                    // ---------- LT2100E register unpack (HMI writes %MW600..609) ----------
// reg[0] button bits: 0=start 1=stop 2=reset 3=ack 4=clean
//                     5=jog+ 6=jog- 7=recipeWrite 8=trimWrite
// Numerics are copied only while their write/jog bit is held, so direct
// variable writes (watch list / sim testing) keep working unchanged.
IF GVL_Cmd.hmiRegsCmd[1] <> 0 THEN
    GVL_Cmd.hmiMaintPin := TO_UINT(GVL_Cmd.hmiRegsCmd[1]);
END_IF
IF (GVL_Cmd.hmiRegsCmd[0] AND 16#0060) <> 0 THEN            // a jog bit is held
    GVL_Cmd.hmiJogAxis := TO_INT(GVL_Cmd.hmiRegsCmd[2]);
END_IF
IF (GVL_Cmd.hmiRegsCmd[0] AND 16#0080) <> 0 THEN            // recipe write
    GVL_Cmd.hmiRecItem  := TO_UINT(GVL_Cmd.hmiRegsCmd[3]);
    GVL_Cmd.hmiRecField := TO_UINT(GVL_Cmd.hmiRegsCmd[4]);
    GVL_Cmd.hmiRecValue := TO_LREAL(GVL_Cmd.hmiRegsCmd[5]) / 10.0;   // x10 scaling
END_IF
IF (GVL_Cmd.hmiRegsCmd[0] AND 16#0100) <> 0 THEN            // trim write
    GVL_Cmd.hmiTrimPress := TO_UINT(GVL_Cmd.hmiRegsCmd[6]);
    GVL_Cmd.hmiTrimDelta := TO_LREAL(TO_INT(GVL_Cmd.hmiRegsCmd[7])) / 100.0;  // x100 signed
END_IF
bJogP := GVL_Cmd.hmiJogPlus  OR ((GVL_Cmd.hmiRegsCmd[0] AND 16#0020) <> 0);
bJogM := GVL_Cmd.hmiJogMinus OR ((GVL_Cmd.hmiRegsCmd[0] AND 16#0040) <> 0);

rtStart(CLK := GVL_Cmd.hmiStart OR ((GVL_Cmd.hmiRegsCmd[0] AND 16#0001) <> 0));
rtStop (CLK := GVL_Cmd.hmiStop  OR ((GVL_Cmd.hmiRegsCmd[0] AND 16#0002) <> 0));
rtReset(CLK := GVL_Cmd.hmiReset OR ((GVL_Cmd.hmiRegsCmd[0] AND 16#0004) <> 0));
rtAck  (CLK := GVL_Cmd.hmiAck   OR ((GVL_Cmd.hmiRegsCmd[0] AND 16#0008) <> 0));
rtClean(CLK := GVL_Cmd.hmiClean OR ((GVL_Cmd.hmiRegsCmd[0] AND 16#0010) <> 0));

GVL_Cmd.reqStart  := rtStart.Q;
GVL_Cmd.reqStop   := rtStop.Q  OR GVL_Cmd.reqStop;    // JobExec may also set; consumed by Supervisor edge
GVL_Cmd.reqReset  := rtReset.Q;
GVL_Cmd.reqAckAll := rtAck.Q;
GVL_Cmd.reqClean  := rtClean.Q OR GVL_Cmd.reqClean;
// self-clearing one-shot semantics: Supervisor uses R_TRIG on these,
// so clear them after one comms cycle
IF NOT rtStop.Q  THEN GVL_Cmd.reqStop  := FALSE; END_IF
IF NOT rtClean.Q THEN GVL_Cmd.reqClean := FALSE; END_IF

// ---------- jog (maintenance only) ----------
jogPermit := (GVL_Cmd.hmiMaintPin = MAINT_PIN)
         AND ((GVL_Sts.mode = E_MachMode.READY) OR (GVL_Sts.mode = E_MachMode.FAULT))
         AND GVL_Sts.safetyOk;
tonJog(IN := jogPermit AND (bJogP OR bJogM), PT := T#100MS);
IF tonJog.Q THEN
    tonJog(IN := FALSE);
    jogStep := LIMIT(1.0, GVL_Par.jogVel, GVL_Cfg.JOG_VEL_MAX) * 0.1;  // mm per 100 ms
    IF bJogM THEN jogStep := -jogStep; END_IF
    CASE GVL_Cmd.hmiJogAxis OF
        1: IF NOT GVL_Mech.axGX.Busy THEN
               GVL_Mech.axGX.TargetPos := GVL_Mech.axGX.Sts.actPos + jogStep;
               GVL_Mech.axGX.Vel := GVL_Par.jogVel;
               GVL_Mech.axGX.MoveExec := TRUE;
           END_IF
        2: IF NOT GVL_Mech.axGT.Busy THEN
               GVL_Mech.axGT.TargetPos := GVL_Mech.axGT.Sts.actPos + jogStep;
               GVL_Mech.axGT.Vel := GVL_Par.jogVel;
               GVL_Mech.axGT.MoveExec := TRUE;
           END_IF
        3: IF NOT GVL_Mech.axGZ.Busy THEN
               GVL_Mech.axGZ.TargetPos := GVL_Mech.axGZ.Sts.actPos + jogStep;
               GVL_Mech.axGZ.Vel := GVL_Par.jogVel;
               GVL_Mech.axGZ.MoveExec := TRUE;
           END_IF
        // axes 4..8: same pattern for scraper X/Y/Z, fork Z/tele — add as needed
    END_CASE
ELSIF NOT (bJogP OR bJogM) THEN
    GVL_Mech.axGX.MoveExec := FALSE;
    GVL_Mech.axGT.MoveExec := FALSE;
    GVL_Mech.axGZ.MoveExec := FALSE;
END_IF

// ---------- recipe editor (bounds-checked; rejected while RUN) ----------
rtRecW(CLK := GVL_Cmd.hmiRecWrite OR ((GVL_Cmd.hmiRegsCmd[0] AND 16#0080) <> 0));
IF rtRecW.Q THEN
    GVL_Cmd.hmiRecAck := FALSE; GVL_Cmd.hmiRecErr := FALSE;
    recIt := TO_INT(GVL_Cmd.hmiRecItem);
    recV  := GVL_Cmd.hmiRecValue;
    recOk := (recIt >= 1) AND (recIt <= 4) AND (GVL_Sts.mode <> E_MachMode.RUN);
    IF recOk THEN
        CASE GVL_Cmd.hmiRecField OF
            1: IF (recV >= GVL_Cfg.REC_COOK_MIN)  AND (recV <= GVL_Cfg.REC_COOK_MAX)
               THEN GVL_Par.aRecipe[recIt].cookTimeS := recV;  ELSE recOk := FALSE; END_IF
            2: IF (recV >= GVL_Cfg.REC_SMDUR_MIN) AND (recV <= GVL_Cfg.REC_SMDUR_MAX)
               THEN GVL_Par.aRecipe[recIt].smashDurS := recV;  ELSE recOk := FALSE; END_IF
            3: IF (recV >= GVL_Cfg.REC_SMPOS_MIN) AND (recV <= GVL_Cfg.REC_SMPOS_MAX)
               THEN GVL_Par.aRecipe[recIt].smashPosMm := recV; ELSE recOk := FALSE; END_IF
            4: IF (recV >= GVL_Cfg.REC_HLPOS_MIN) AND (recV <= GVL_Cfg.REC_HLPOS_MAX)
               THEN GVL_Par.aRecipe[recIt].holdPosMm := recV;  ELSE recOk := FALSE; END_IF
            5: IF (recV >= GVL_Cfg.REC_PLSET_MIN) AND (recV <= GVL_Cfg.REC_PLSET_MAX)
               THEN GVL_Par.aRecipe[recIt].platenSetC := recV; ELSE recOk := FALSE; END_IF
        ELSE
            recOk := FALSE;
        END_CASE
        // physical sanity: hold gap must not be tighter than smash gap
        IF recOk AND (GVL_Par.aRecipe[recIt].holdPosMm < GVL_Par.aRecipe[recIt].smashPosMm) THEN
            GVL_Par.aRecipe[recIt].holdPosMm := GVL_Par.aRecipe[recIt].smashPosMm;
        END_IF
    END_IF
    GVL_Cmd.hmiRecAck := recOk;
    GVL_Cmd.hmiRecErr := NOT recOk;
END_IF

// ---------- press calibration trim (maintenance PIN; not while RUN) ----------
rtTrimW(CLK := GVL_Cmd.hmiTrimWrite OR ((GVL_Cmd.hmiRegsCmd[0] AND 16#0100) <> 0));
IF rtTrimW.Q THEN
    GVL_Cmd.hmiTrimAck := FALSE; GVL_Cmd.hmiTrimErr := FALSE;
    trimP := TO_INT(GVL_Cmd.hmiTrimPress);
    IF (trimP >= 0) AND (trimP <= 3)
       AND (GVL_Cmd.hmiMaintPin = MAINT_PIN)
       AND (GVL_Sts.mode <> E_MachMode.RUN)
       AND (ABS(GVL_Cmd.hmiTrimDelta) <= GVL_Cfg.PRESS_TRIM_MAX_MM) THEN
        GVL_Par.pressTrimMm[trimP] := LIMIT(-GVL_Cfg.PRESS_TRIM_MAX_MM,
            GVL_Par.pressTrimMm[trimP] + GVL_Cmd.hmiTrimDelta,
            GVL_Cfg.PRESS_TRIM_MAX_MM);
        GVL_Cmd.hmiTrimAck := TRUE;
    ELSE
        GVL_Cmd.hmiTrimErr := TRUE;
    END_IF
END_IF

// ---------- LT2100E status pack (HMI reads %MW620..669) ----------
GVL_Cmd.hmiRegsSts[0] := TO_WORD(TO_UINT(GVL_Sts.mode));
wFlags := 0;
IF GVL_Cmd.hmiRecAck    THEN wFlags := wFlags OR 16#0001; END_IF
IF GVL_Cmd.hmiRecErr    THEN wFlags := wFlags OR 16#0002; END_IF
IF GVL_Cmd.hmiTrimAck   THEN wFlags := wFlags OR 16#0004; END_IF
IF GVL_Cmd.hmiTrimErr   THEN wFlags := wFlags OR 16#0008; END_IF
IF GVL_Sts.heatAtSet    THEN wFlags := wFlags OR 16#0010; END_IF
IF GVL_Sts.fridgeAtSet  THEN wFlags := wFlags OR 16#0020; END_IF
IF GVL_Sts.allHomed     THEN wFlags := wFlags OR 16#0040; END_IF
IF GVL_Sts.safetyOk     THEN wFlags := wFlags OR 16#0080; END_IF
IF GVL_Sts.cleanCoolOk  THEN wFlags := wFlags OR 16#0100; END_IF
GVL_Cmd.hmiRegsSts[1] := wFlags;
GVL_Cmd.hmiRegsSts[2] := TO_WORD(TO_UINT(GVL_Alm.nActive));
GVL_Cmd.hmiRegsSts[3] := TO_WORD(GVL_Alm.aActive[0].id AND 16#FFFF);          // code
GVL_Cmd.hmiRegsSts[4] := TO_WORD(SHR(GVL_Alm.aActive[0].id, 16) AND 16#FFFF); // subsystem
GVL_Cmd.hmiRegsSts[5] := TO_WORD(TO_UINT(GVL_Sts.uptimeS MOD 65536));
// griddle states 626..629
FOR z2 := 0 TO 3 DO
    GVL_Cmd.hmiRegsSts[6 + z2] := TO_WORD(GVL_Sts.aGriddle[z2].state);
END_FOR
// recipe readback 630..649: per item 1..4 -> cook, smashDur, smashPos, holdPos, platenSet (all x10)
FOR it2 := 1 TO 4 DO
    base := 10 + (it2 - 1) * 5;
    GVL_Cmd.hmiRegsSts[base]     := TO_WORD(TO_UINT(GVL_Par.aRecipe[it2].cookTimeS  * 10.0));
    GVL_Cmd.hmiRegsSts[base + 1] := TO_WORD(TO_UINT(GVL_Par.aRecipe[it2].smashDurS  * 10.0));
    GVL_Cmd.hmiRegsSts[base + 2] := TO_WORD(TO_UINT(GVL_Par.aRecipe[it2].smashPosMm * 10.0));
    GVL_Cmd.hmiRegsSts[base + 3] := TO_WORD(TO_UINT(GVL_Par.aRecipe[it2].holdPosMm  * 10.0));
    GVL_Cmd.hmiRegsSts[base + 4] := TO_WORD(TO_UINT(GVL_Par.aRecipe[it2].platenSetC * 10.0));
END_FOR
// press trims 650..653 (x100 signed)
FOR z2 := 0 TO 3 DO
    GVL_Cmd.hmiRegsSts[30 + z2] := TO_WORD(TO_INT(GVL_Par.pressTrimMm[z2] * 100.0));
END_FOR
// temperatures 654..661 platens, 662 fridge (x10)
FOR z2 := 0 TO 7 DO
    GVL_Cmd.hmiRegsSts[34 + z2] := TO_WORD(TO_INT(GVL_Sts.aHeat[z2].actC * 10.0));
END_FOR
GVL_Cmd.hmiRegsSts[42] := TO_WORD(TO_INT(GVL_Sts.fridgeActC * 10.0));

                  
END_PROGRAM

(* ============================================================ PRG_Carousels — T_App body-call owner: press drives, presses, pneumatics, VFD indexers, carousels, airlock. Pure wiring (the ST equivalent of a CFC sheet). Runs AFTER Supervisor/ JobExec/Test (which write the Cmd inputs). ============================================================ *)
PROGRAM PRG_Carousels
  VAR
    i : INT;
    init : BOOL;
  END_VAR

                    IF NOT init THEN
    init := TRUE;
    FOR i := 0 TO 3 DO
        GVL_Mech.drvPress[i].SubsysId := GVL_Cfg.SS_PRESS_0 + TO_UINT(i);
        GVL_Mech.fbPress[i].PressId := i;
    END_FOR
    GVL_Mech.fbDoorFridgeFront.SubsysId := GVL_Cfg.SS_AIRLOCK;
    GVL_Mech.fbDoorFridgeSide.SubsysId  := GVL_Cfg.SS_AIRLOCK;
    GVL_Mech.fbDoorChamber.SubsysId     := GVL_Cfg.SS_AIRLOCK;
    GVL_Mech.fbPinGriddle.SubsysId := GVL_Cfg.SS_GRID_CAR;
    GVL_Mech.fbPinFridge.SubsysId  := GVL_Cfg.SS_FRIDGE_CAR;
    GVL_Mech.fbPneuGrip.SubsysId   := GVL_Cfg.SS_GRIPPER;
    GVL_Mech.vfdGriddle.SubsysId := GVL_Cfg.SS_GRID_CAR;
    GVL_Mech.vfdFridge.SubsysId  := GVL_Cfg.SS_FRIDGE_CAR;
END_IF

// ---- presses ----
FOR i := 0 TO 3 DO
    GVL_Mech.fbPress[i].Enable := GVL_Sts.enMotion;
    GVL_Mech.fbPress[i].Abort  := GVL_Sts.abortAll;
    GVL_Mech.fbPress[i].Sim    := GVL_Cfg.SIM_MODE;
    GVL_Mech.fbPress[i].CycleMs:= GVL_Cfg.T_APP_MS;
    // bench override: the selected drive runs REAL while the machine is sim
    GVL_Mech.drvPress[i].Sim    := GVL_Cfg.SIM_MODE AND (i <> GVL_Cfg.PRESS_BENCH_DRIVE);
    GVL_Mech.drvPress[i].Enable := GVL_Sts.enMotion;
    GVL_Mech.drvPress[i].Abort  := GVL_Sts.abortAll;
    GVL_Mech.drvPress[i].CycleMs:= GVL_Cfg.T_APP_MS;
    GVL_Mech.drvPress[i].iInPos := GVL_IO.iPressInPos[i];
    GVL_Mech.drvPress[i].iAlarm := GVL_IO.iPressAlarm[i];
    GVL_Mech.fbPress[i](Drv := GVL_Mech.drvPress[i]);
    GVL_Mech.drvPress[i]();
    IF (NOT GVL_Cfg.SIM_MODE) OR (i = GVL_Cfg.PRESS_BENCH_DRIVE) THEN
        GVL_IO.qPressSel0[i]   := GVL_Mech.drvPress[i].qSel0;
        GVL_IO.qPressSel1[i]   := GVL_Mech.drvPress[i].qSel1;
        GVL_IO.qPressCtrg[i]   := GVL_Mech.drvPress[i].qCtrg;
        GVL_IO.qPressEnable[i] := GVL_Mech.drvPress[i].qEnable;
    END_IF
END_FOR

// ---- CS2RS Modbus PR-write transport: NetworkConfig channel routing ----
// Channels are created in NetworkConfig (RS485 -> Modbus Master), one
// write-multiple channel per PR path (see GVL_IO placeholders + GVL_Cfg
// reference). This glue routes the bench/press-0 drive's path-write request
// to the matching channel. Extend with channel banks for drives 1..3 when
// the full RS485 bus exists.
IF (NOT GVL_Cfg.SIM_MODE) OR (GVL_Cfg.PRESS_BENCH_DRIVE >= 0) THEN
    GVL_IO.qMbPr0Trig := FALSE;
    GVL_IO.qMbPr1Trig := FALSE;
    GVL_IO.qMbPr2Trig := FALSE;
    GVL_Mech.drvPress[0].MbWrDone := FALSE;
    GVL_Mech.drvPress[0].MbWrErr  := FALSE;
    CASE GVL_Mech.drvPress[0].MbPath OF
        0:  GVL_IO.qMbPr0Data[0] := GVL_Mech.drvPress[0].MbValH;
            GVL_IO.qMbPr0Data[1] := GVL_Mech.drvPress[0].MbValL;
            GVL_IO.qMbPr0Trig    := GVL_Mech.drvPress[0].MbWrExec;
            GVL_Mech.drvPress[0].MbWrDone := GVL_IO.iMbPr0Done AND GVL_Mech.drvPress[0].MbWrExec;
        1:  GVL_IO.qMbPr1Data[0] := GVL_Mech.drvPress[0].MbValH;
            GVL_IO.qMbPr1Data[1] := GVL_Mech.drvPress[0].MbValL;
            GVL_IO.qMbPr1Trig    := GVL_Mech.drvPress[0].MbWrExec;
            GVL_Mech.drvPress[0].MbWrDone := GVL_IO.iMbPr1Done AND GVL_Mech.drvPress[0].MbWrExec;
        2:  GVL_IO.qMbPr2Data[0] := GVL_Mech.drvPress[0].MbValH;
            GVL_IO.qMbPr2Data[1] := GVL_Mech.drvPress[0].MbValL;
            GVL_IO.qMbPr2Trig    := GVL_Mech.drvPress[0].MbWrExec;
            GVL_Mech.drvPress[0].MbWrDone := GVL_IO.iMbPr2Done AND GVL_Mech.drvPress[0].MbWrExec;
    END_CASE
    GVL_Mech.drvPress[0].MbWrErr :=
        (GVL_IO.iMbPrErr <> 0) AND GVL_Mech.drvPress[0].MbWrExec;
END_IF

// ---- pneumatics ----
GVL_Mech.fbDoorFridgeSide(Sim := GVL_Cfg.SIM_MODE, CycleMs := GVL_Cfg.T_APP_MS,
    iExtended := GVL_IO.iDoorFrSide_Op, iRetracted := GVL_IO.iDoorFrSide_Cl);
GVL_Mech.fbDoorChamber(Sim := GVL_Cfg.SIM_MODE, CycleMs := GVL_Cfg.T_APP_MS,
    iExtended := GVL_IO.iDoorChamber_Op, iRetracted := GVL_IO.iDoorChamber_Cl);
GVL_Mech.fbDoorFridgeFront(Sim := GVL_Cfg.SIM_MODE, CycleMs := GVL_Cfg.T_APP_MS,
    iExtended := GVL_IO.iDoorFrFront_Op, iRetracted := GVL_IO.iDoorFrFront_Cl);
GVL_Mech.fbPinGriddle(Sim := GVL_Cfg.SIM_MODE, CycleMs := GVL_Cfg.T_APP_MS,
    iExtended := GVL_IO.iPinGriddle_Ext, iRetracted := GVL_IO.iPinGriddle_Ret);
GVL_Mech.fbPinFridge(Sim := GVL_Cfg.SIM_MODE, CycleMs := GVL_Cfg.T_APP_MS,
    iExtended := GVL_IO.iPinFridge_Ext, iRetracted := GVL_IO.iPinFridge_Ret);
GVL_Mech.fbPneuGrip(Sim := GVL_Cfg.SIM_MODE, CycleMs := GVL_Cfg.T_APP_MS,
    iExtended := GVL_IO.iGripAcquired, iRetracted := NOT GVL_IO.iGripAcquired);
IF NOT GVL_Cfg.SIM_MODE THEN
    GVL_IO.qDoorFridgeSide  := GVL_Mech.fbDoorFridgeSide.qValve;
    GVL_IO.qDoorChamber     := GVL_Mech.fbDoorChamber.qValve;
    GVL_IO.qDoorFridgeFront := GVL_Mech.fbDoorFridgeFront.qValve;
    GVL_IO.qPinGriddle      := GVL_Mech.fbPinGriddle.qValve;
    GVL_IO.qPinFridge       := GVL_Mech.fbPinFridge.qValve;
    GVL_IO.qGripper         := GVL_Mech.fbPneuGrip.qValve;
END_IF

// ---- airlock ----
GVL_Mech.fbAirlock(
    Enable := GVL_Sts.enMotion, Abort := GVL_Sts.abortAll,
    DoorFridge := GVL_Mech.fbDoorFridgeSide,
    DoorChamber := GVL_Mech.fbDoorChamber);

// ---- carousels ----
GVL_Mech.vfdGriddle.Sim := GVL_Cfg.SIM_MODE;  GVL_Mech.vfdGriddle.CycleMs := GVL_Cfg.T_APP_MS;
GVL_Mech.vfdGriddle.iEnc := GVL_IO.diGridCarEnc;
GVL_Mech.vfdGriddle.iHomeProx := GVL_IO.iGridCarHome;
GVL_Mech.vfdFridge.Sim := GVL_Cfg.SIM_MODE;   GVL_Mech.vfdFridge.CycleMs := GVL_Cfg.T_APP_MS;
GVL_Mech.vfdFridge.iEnc := GVL_IO.diFrCarEnc;
GVL_Mech.vfdFridge.iHomeProx := GVL_IO.iFrCarHome;

GVL_Mech.fbGridCar(
    Enable := GVL_Sts.enMotion, Abort := GVL_Sts.abortAll,
    Vfd := GVL_Mech.vfdGriddle, Pin := GVL_Mech.fbPinGriddle);
GVL_Mech.fbFridgeCar(
    Enable := GVL_Sts.enMotion, Abort := GVL_Sts.abortAll,
    Vfd := GVL_Mech.vfdFridge, Pin := GVL_Mech.fbPinFridge);
GVL_Mech.vfdGriddle();
GVL_Mech.vfdFridge();
IF NOT GVL_Cfg.SIM_MODE THEN
    GVL_IO.qGridCarFwd := GVL_Mech.vfdGriddle.qFwd;
    GVL_IO.qGridCarRev := GVL_Mech.vfdGriddle.qRev;
    GVL_IO.wGridCarSpeed := GVL_Mech.vfdGriddle.qSpeed;
    GVL_IO.qFrCarFwd := GVL_Mech.vfdFridge.qFwd;
    GVL_IO.qFrCarRev := GVL_Mech.vfdFridge.qRev;
    GVL_IO.wFrCarSpeed := GVL_Mech.vfdFridge.qSpeed;
END_IF
GVL_Sts.carGridStation := GVL_Mech.fbGridCar.ActStation;
GVL_Sts.carFridgeFace  := GVL_Mech.fbFridgeCar.ActFace;


                  
END_PROGRAM

(* ============================================================ PRG_Heating — T_App body-call owner: 8 heaters + bank + fridge. Zone map: griddle g -> zones 2g (top), 2g+1 (bottom). Setpoint follows the active recipe of the griddle's item; empty griddles idle at the BEEF setpoint so they are ready to load. ============================================================ *)
PROGRAM PRG_Heating
  VAR
    z : INT;
    g : INT;
    itm : UINT;
    setC : LREAL;
  END_VAR

                    FOR z := 0 TO 7 DO
    g := z / 2;
    itm := GVL_Sts.aGriddle[g].item;
    IF itm = 0 THEN itm := 1; END_IF          // idle at BEEF setpoint
    setC := GVL_Par.aRecipe[itm].platenSetC;
    GVL_Mech.fbHeater[z].Sim := GVL_Cfg.SIM_MODE;
    GVL_Mech.fbHeater[z].ZoneId := z;
    GVL_Mech.fbHeater[z].CycleMs := GVL_Cfg.T_APP_MS;
    GVL_Mech.fbHeater[z].Enable := GVL_Sts.enProcess;
    GVL_Mech.fbHeater[z].SetC := setC;
    GVL_Mech.fbHeater[z].iTempRaw := GVL_IO.wPlatenTemp[z];
    GVL_Mech.fbHeater[z].StaggerToken := GVL_Mech.fbHeatBank.Token[z];
    GVL_Mech.fbHeater[z]();
    IF NOT GVL_Cfg.SIM_MODE THEN
        GVL_IO.qSsr[z] := GVL_Mech.fbHeater[z].qSsr;
    END_IF
    GVL_Sts.aHeat[z] := GVL_Mech.fbHeater[z].Zone;
END_FOR
GVL_Mech.fbHeatBank(Enable := GVL_Sts.enProcess, Heaters := GVL_Mech.fbHeater);

GVL_Mech.fbRefrig(
    Sim := GVL_Cfg.SIM_MODE,
    Enable := GVL_Sts.enProcess,
    iTempRaw := GVL_IO.wFridgeTemp,
    CycleMs := GVL_Cfg.T_APP_MS);
// (compressor output relay would be copied to GVL_IO here at migration)


                  
END_PROGRAM

(* ============================================================ PRG_IoMap — T_App, runs FIRST. Housekeeping + the place for commissioning force-rungs (these networks become LD at the language refactor). All %I/%Q symbol reads/writes elsewhere go through the owner wiring PRGs; addresses exist ONLY in GVL_IO. ============================================================ *)
PROGRAM PRG_IoMap
  VAR
    msAcc : LREAL;
  END_VAR

                    msAcc := msAcc + GVL_Cfg.T_APP_MS;
IF msAcc >= 1000.0 THEN
    msAcc := msAcc - 1000.0;
    GVL_Sts.uptimeS := GVL_Sts.uptimeS + 1;
END_IF
// ---- bench press-drive terminal mapping (active when PRESS_BENCH_DRIVE = 0) ----
// Copies the unaddressed press-0 signal arrays to/from the physically wired
// bench terminals (declared in GVL_IO, old-rig addresses).
IF GVL_Cfg.PRESS_BENCH_DRIVE = 0 THEN
    GVL_IO.qBenchPrAdd0    := GVL_IO.qPressSel0[0];
    GVL_IO.qBenchPrAdd1    := GVL_IO.qPressSel1[0];
    GVL_IO.qBenchPrCtrg    := GVL_IO.qPressCtrg[0];
    GVL_IO.qBenchPrDisable := NOT GVL_IO.qPressEnable[0];   // wire is a DISABLE line
    GVL_IO.iPressInPos[0]  := GVL_IO.iBenchPrInPos;
    GVL_IO.iPressAlarm[0]  := GVL_IO.iBenchPrAlarm;         // if ALM is NC: invert here
END_IF

// TODO(commissioning): add per-signal force flags here, e.g.
//   IF forceDoorChamber THEN GVL_IO.qDoorChamber := forceVal; END_IF
                  
END_PROGRAM

(* ============================================================ PRG_Motion — T_Motion (4 ms). Body-call owner for all axis FBs and the motion mechanisms. THE ONLY TASK TOUCHING MC_* / AXIS_REF. This is the ST equivalent of the CFC wiring diagram: pure parameter assignment + instance calls, no logic. MIGRATION: replace GVL_Axes.axRef* with the device-tree axis objects created by the EtherCAT scan (step 3 of the guide). ============================================================ *)
PROGRAM PRG_Motion
  VAR
    init : BOOL;
  END_VAR

                    IF NOT init THEN
    init := TRUE;
    GVL_Mech.axGX.SubsysId := GVL_Cfg.SS_GANTRY_X;   GVL_Mech.axGX.CycleMs := GVL_Cfg.T_MOTION_MS;
    GVL_Mech.axGT.SubsysId := GVL_Cfg.SS_GANTRY_T;   GVL_Mech.axGT.CycleMs := GVL_Cfg.T_MOTION_MS;
    GVL_Mech.axGZ.SubsysId := GVL_Cfg.SS_GANTRY_Z;   GVL_Mech.axGZ.CycleMs := GVL_Cfg.T_MOTION_MS;
    GVL_Mech.axSX.SubsysId := GVL_Cfg.SS_SCRAPER_X;  GVL_Mech.axSX.CycleMs := GVL_Cfg.T_MOTION_MS;
    GVL_Mech.axSY.SubsysId := GVL_Cfg.SS_SCRAPER_Y;  GVL_Mech.axSY.CycleMs := GVL_Cfg.T_MOTION_MS;
    GVL_Mech.axSZ.SubsysId := GVL_Cfg.SS_SCRAPER_Z;  GVL_Mech.axSZ.CycleMs := GVL_Cfg.T_MOTION_MS;
    GVL_Mech.axFZ.SubsysId := GVL_Cfg.SS_FORK_Z;     GVL_Mech.axFZ.CycleMs := GVL_Cfg.T_MOTION_MS;
    GVL_Mech.axFT.SubsysId := GVL_Cfg.SS_FORK_TELE;  GVL_Mech.axFT.CycleMs := GVL_Cfg.T_MOTION_MS;
END_IF

// ---- distribute enables / abort / reset ----
GVL_Mech.axGX.Sim := GVL_Cfg.SIM_MODE;  GVL_Mech.axGX.Enable := GVL_Sts.enMotion;
GVL_Mech.axGT.Sim := GVL_Cfg.SIM_MODE;  GVL_Mech.axGT.Enable := GVL_Sts.enMotion;
GVL_Mech.axGZ.Sim := GVL_Cfg.SIM_MODE;  GVL_Mech.axGZ.Enable := GVL_Sts.enMotion;
GVL_Mech.axSX.Sim := GVL_Cfg.SIM_MODE;  GVL_Mech.axSX.Enable := GVL_Sts.enMotion;
GVL_Mech.axSY.Sim := GVL_Cfg.SIM_MODE;  GVL_Mech.axSY.Enable := GVL_Sts.enMotion;
GVL_Mech.axSZ.Sim := GVL_Cfg.SIM_MODE;  GVL_Mech.axSZ.Enable := GVL_Sts.enMotion;
GVL_Mech.axFZ.Sim := GVL_Cfg.SIM_MODE;  GVL_Mech.axFZ.Enable := GVL_Sts.enMotion;
GVL_Mech.axFT.Sim := GVL_Cfg.SIM_MODE;  GVL_Mech.axFT.Enable := GVL_Sts.enMotion;
GVL_Mech.axGX.Abort := GVL_Sts.abortAll;  GVL_Mech.axGX.ResetExec := GVL_Sts.resetPulse;
GVL_Mech.axGT.Abort := GVL_Sts.abortAll;  GVL_Mech.axGT.ResetExec := GVL_Sts.resetPulse;
GVL_Mech.axGZ.Abort := GVL_Sts.abortAll;  GVL_Mech.axGZ.ResetExec := GVL_Sts.resetPulse;
GVL_Mech.axSX.Abort := GVL_Sts.abortAll;  GVL_Mech.axSX.ResetExec := GVL_Sts.resetPulse;
GVL_Mech.axSY.Abort := GVL_Sts.abortAll;  GVL_Mech.axSY.ResetExec := GVL_Sts.resetPulse;
GVL_Mech.axSZ.Abort := GVL_Sts.abortAll;  GVL_Mech.axSZ.ResetExec := GVL_Sts.resetPulse;
GVL_Mech.axFZ.Abort := GVL_Sts.abortAll;  GVL_Mech.axFZ.ResetExec := GVL_Sts.resetPulse;
GVL_Mech.axFT.Abort := GVL_Sts.abortAll;  GVL_Mech.axFT.ResetExec := GVL_Sts.resetPulse;

// ---- mechanism bodies (write axis inputs) ----
GVL_Mech.fbGripper(
    Sim  := GVL_Cfg.SIM_MODE,
    iAcquired := GVL_IO.iGripAcquired,
    Pneu := GVL_Mech.fbPneuGrip);

GVL_Mech.fbGantry(
    Enable := GVL_Sts.enMotion,
    Abort  := GVL_Sts.abortAll,
    Sim    := GVL_Cfg.SIM_MODE,
    AxX := GVL_Mech.axGX, AxT := GVL_Mech.axGT, AxZ := GVL_Mech.axGZ,
    Grip := GVL_Mech.fbGripper, IK := GVL_Mech.fbIK);

GVL_Mech.fbScraper(
    Enable := GVL_Sts.enMotion,
    Abort  := GVL_Sts.abortAll,
    Sim    := GVL_Cfg.SIM_MODE,
    AxX := GVL_Mech.axSX, AxY := GVL_Mech.axSY, AxZ := GVL_Mech.axSZ);

GVL_Mech.fbFork(
    Enable := GVL_Sts.enMotion,
    Abort  := GVL_Sts.abortAll,
    Sim    := GVL_Cfg.SIM_MODE,
    iBrakeOk := GVL_IO.iForkBrakeOk,
    iTrayPresent := GVL_IO.iForkTrayPresent,
    AxZ := GVL_Mech.axFZ, AxT := GVL_Mech.axFT);
IF NOT GVL_Cfg.SIM_MODE THEN
    GVL_IO.qForkBrakeRelease := GVL_Mech.fbFork.qBrakeRelease;
END_IF

// ---- axis bodies LAST (consume inputs written above) ----
GVL_Mech.axGX(Axis := GVL_Axes.axRefGantryX);
GVL_Mech.axGT(Axis := GVL_Axes.axRefGantryT);
GVL_Mech.axGZ(Axis := GVL_Axes.axRefGantryZ);
GVL_Mech.axSX(Axis := GVL_Axes.axRefScraperX);
GVL_Mech.axSY(Axis := GVL_Axes.axRefScraperY);
GVL_Mech.axSZ(Axis := GVL_Axes.axRefScraperZ);
GVL_Mech.axFZ(Axis := GVL_Axes.axRefForkZ);
GVL_Mech.axFT(Axis := GVL_Axes.axRefForkTele);


                  
END_PROGRAM

(* ============================================================ PRG_Sim — T_App. Plant models beyond what L1 drivers model internally. v1: reserved (axis/pneu/thermal/fridge models are inside their driver FBs; patty bookkeeping is in JobExec). Extend here for: patty-present optics model, condensation / door-open thermal coupling, disturbance injection. ============================================================ *)
PROGRAM PRG_Sim

                    ;
                  
END_PROGRAM

(* ============================================================ PRG_Test — automated regression suite (T_App, after JobExec). Start: set GVL_Cmd.testStart := TRUE (rising edge) once mode has reached READY. Results: aResult[n] : 0=pending 1=PASS 2=FAIL (n = 1..10) aFailCode[n] : diagnostic (step*1000 or ErrorID low word) PassCount / suiteDone TC list: 1 boot->READY + allHomed 6 griddle carousel 1,3,0 2 IK table (24 pick + 6 place) 7 fork fetch/return L5 3 heat AtSet + fridge + stagger 8 gantry pick/place/park 4 airlock mutual exclusion 9 full cycle via Gateway regs 5 press smash->hold->open 10 fault inject + recovery x2 ============================================================ *)
PROGRAM PRG_Test
  VAR
    aResult : ARRAY[1..10] OF INT;
    aFailCode : ARRAY[1..10] OF UDINT;
    PassCount : INT;
    suiteDone : BOOL;
    running : BOOL;
    tc : INT;  (* current test case *)
    stp : INT;  (* step within test case *)
    rtStart : R_TRIG;
    tonG : TON;  (* per-step guard timer *)
    ptCur : TIME;
    i : INT;
    k : INT;
    px : LREAL;  (* TC2 locals *)
    py : LREAL;
    xr : LREAL;
    yr : LREAL;
    thR : LREAL;
    ikFail : BOOL;
    nRamp : INT;  (* TC3 locals *)
    stagViol : BOOL;
    testSeq : UINT;  (* TC9 locals *)
    hbCnt : UINT;
    hbDiv : INT;
    haccp0 : UDINT;
    holdCnt : INT;
    PI_ : LREAL := 3.14159265358979;
  END_VAR

                    rtStart(CLK := GVL_Cmd.testStart);
IF rtStart.Q AND NOT running THEN
    running := TRUE; suiteDone := FALSE;
    FOR i := 1 TO 10 DO aResult[i] := 0; aFailCode[i] := 0; END_FOR
    PassCount := 0;
    tc := 1; stp := 0;
END_IF
IF NOT running THEN RETURN; END_IF

// keep simulated gateway heartbeat alive during the whole suite
hbDiv := hbDiv + 1;
IF hbDiv >= 25 THEN   // every 500 ms
    hbDiv := 0; hbCnt := hbCnt + 1;
    GVL_Cmd.mbCmdRegs[9] := hbCnt;
END_IF

// per-step guard
tonG(IN := TRUE, PT := ptCur);

CASE tc OF
// ================= TC1: boot -> READY =================
1:
    CASE stp OF
        0: ptCur := T#90S; tonG(IN := FALSE); stp := 1;
        1:
            IF (GVL_Sts.mode = E_MachMode.READY) AND GVL_Sts.allHomed THEN
                aResult[1] := 1; tc := 2; stp := 0;
            ELSIF tonG.Q THEN
                aResult[1] := 2; aFailCode[1] := TO_UDINT(TO_UINT(GVL_Sts.mode));
                tc := 2; stp := 0;
            END_IF
    END_CASE

// ================= TC2: IK table =================
2:
    ikFail := FALSE;
    FOR i := 0 TO GVL_Cfg.PATTIES_PER_TRAY - 1 DO
        px := GVL_Cfg.PICK_BASE_X + TO_LREAL(i MOD GVL_Cfg.TRAY_COLS) * GVL_Cfg.PICK_SPACING_X;
        py := GVL_Cfg.PICK_BASE_Y + TO_LREAL(i / GVL_Cfg.TRAY_COLS) * GVL_Cfg.PICK_SPACING_Y;
        GVL_Mech.fbIK(xCart := px, yCart := py);
        IF NOT GVL_Mech.fbIK.Reachable THEN ikFail := TRUE; aFailCode[2] := TO_UDINT(TO_UINT(i)); END_IF
        thR := GVL_Mech.fbIK.thetaDeg * PI_ / 180.0;
        xr := GVL_Mech.fbIK.xLin + GVL_Cfg.ARM_LEN * COS(thR);
        yr := GVL_Cfg.ARM_LEN * SIN(thR);
        IF (ABS(xr - px) > 0.01) OR (ABS(yr - py) > 0.01) THEN
            ikFail := TRUE; aFailCode[2] := 1000 + TO_UDINT(TO_UINT(i));
        END_IF
    END_FOR
    FOR i := 0 TO GVL_Cfg.PATTIES_PER_GRIDDLE - 1 DO
        px := GVL_Cfg.PLACE_BASE_X + TO_LREAL(i MOD GVL_Cfg.PLACE_COLS) * GVL_Cfg.PLACE_SPC_X;
        py := GVL_Cfg.PLACE_BASE_Y + TO_LREAL(i / GVL_Cfg.PLACE_COLS) * GVL_Cfg.PLACE_SPC_Y;
        GVL_Mech.fbIK(xCart := px, yCart := py);
        IF NOT GVL_Mech.fbIK.Reachable THEN ikFail := TRUE; aFailCode[2] := 2000 + TO_UDINT(TO_UINT(i)); END_IF
    END_FOR
    IF ikFail THEN aResult[2] := 2; ELSE aResult[2] := 1; END_IF
    tc := 3; stp := 0;

// ================= TC3: heat + fridge + stagger =================
3:
    CASE stp OF
        0: ptCur := T#240S; tonG(IN := FALSE); stagViol := FALSE; stp := 1;
        1:
            // stagger monitor: count zones actively ramping WITH token
            nRamp := 0;
            FOR i := 0 TO 7 DO
                IF GVL_Mech.fbHeatBank.Token[i]
                   AND ((GVL_Sts.aHeat[i].setC - GVL_Sts.aHeat[i].actC) > 20.0) THEN
                    nRamp := nRamp + 1;
                END_IF
            END_FOR
            IF nRamp > GVL_Cfg.HEAT_MAX_STAGGER THEN stagViol := TRUE; END_IF
            IF GVL_Sts.heatAtSet AND GVL_Sts.fridgeAtSet THEN
                IF stagViol THEN aResult[3] := 2; aFailCode[3] := 1;
                ELSE aResult[3] := 1; END_IF
                tc := 4; stp := 0;
            ELSIF tonG.Q THEN
                aResult[3] := 2; aFailCode[3] := 2;
                tc := 4; stp := 0;
            END_IF
    END_CASE

// ================= TC4: airlock mutual exclusion =================
4:
    CASE stp OF
        0:
            ptCur := T#10S; tonG(IN := FALSE);
            GVL_Mech.fbAirlock.ReqFridgeOpen := TRUE;
            stp := 1;
        1:
            IF GVL_Mech.fbAirlock.FridgeOpen THEN
                GVL_Mech.fbAirlock.ReqChamberOpen := TRUE;  // request BOTH
                tonG(IN := FALSE); stp := 2;
            ELSIF tonG.Q THEN stp := 90; END_IF
        2: // hold both requests 2 s; invariant must hold
            IF GVL_Mech.fbAirlock.FridgeOpen AND GVL_Mech.fbAirlock.ChamberOpen THEN stp := 90; END_IF
            IF tonG.ET >= T#2S THEN
                GVL_Mech.fbAirlock.ReqFridgeOpen := FALSE;   // yield to chamber
                tonG(IN := FALSE); stp := 3;
            END_IF
        3:
            IF GVL_Mech.fbAirlock.FridgeOpen AND GVL_Mech.fbAirlock.ChamberOpen THEN stp := 90; END_IF
            IF GVL_Mech.fbAirlock.ChamberOpen THEN
                GVL_Mech.fbAirlock.ReqChamberOpen := FALSE;
                tonG(IN := FALSE); stp := 4;
            ELSIF tonG.Q THEN stp := 90; END_IF
        4:
            IF GVL_Mech.fbAirlock.ChamberSealed THEN
                aResult[4] := 1; tc := 5; stp := 0;
            ELSIF tonG.Q THEN stp := 90; END_IF
        90:
            GVL_Mech.fbAirlock.ReqFridgeOpen := FALSE;
            GVL_Mech.fbAirlock.ReqChamberOpen := FALSE;
            aResult[4] := 2; aFailCode[4] := TO_UDINT(TO_UINT(stp));
            tc := 5; stp := 0;
    END_CASE

// ================= TC5: press profile =================
5:
    CASE stp OF
        0:
            ptCur := T#20S; tonG(IN := FALSE);
            GVL_Mech.fbPress[0].Recipe := GVL_Par.aRecipe[1];   // BEEF
            GVL_Mech.fbPress[0].Cmd.code := GVL_Cfg.MCMD_PROFILE;
            GVL_Mech.fbPress[0].CmdExec := TRUE;
            stp := 1;
        1:
            IF GVL_Mech.fbPress[0].Holding THEN
                GVL_Mech.fbPress[0].CmdExec := FALSE;
                IF GVL_Mech.fbPress[0].DwellS < GVL_Par.aRecipe[1].smashDurS - 1.0 THEN
                    aFailCode[5] := 1; stp := 90;
                ELSE
                    GVL_Mech.fbPress[0].Cmd.code := GVL_Cfg.MCMD_OPEN;
                    tonG(IN := FALSE); stp := 12;   // one-scan gap: R_TRIG needs FALSE->TRUE across scans
                END_IF
            ELSIF GVL_Mech.fbPress[0].Error OR tonG.Q THEN
                GVL_Mech.fbPress[0].CmdExec := FALSE;
                aFailCode[5] := GVL_Mech.fbPress[0].ErrorID; stp := 90;
            END_IF
        12: // re-arm on a fresh scan
            GVL_Mech.fbPress[0].CmdExec := TRUE;
            stp := 2;
        2:
            IF GVL_Mech.fbPress[0].IsOpen THEN
                GVL_Mech.fbPress[0].CmdExec := FALSE;
                aResult[5] := 1; tc := 6; stp := 0;
            ELSIF GVL_Mech.fbPress[0].Error OR tonG.Q THEN
                GVL_Mech.fbPress[0].CmdExec := FALSE;
                aFailCode[5] := GVL_Mech.fbPress[0].ErrorID; stp := 90;
            END_IF
        90:
            aResult[5] := 2; tc := 6; stp := 0;
    END_CASE

// ================= TC6: griddle carousel =================
6:
    CASE stp OF
        0: // park gantry first so rotation permissive is TRUE
            ptCur := T#20S; tonG(IN := FALSE);
            GVL_Mech.fbGantry.Cmd.code := GVL_Cfg.MCMD_PARK;
            GVL_Mech.fbGantry.CmdExec := TRUE;
            stp := 1;
        1:
            IF GVL_Mech.fbGantry.Done AND GVL_Mech.fbGantry.Parked THEN
                GVL_Mech.fbGantry.CmdExec := FALSE; k := 0;
                tonG(IN := FALSE); stp := 2;
            ELSIF GVL_Mech.fbGantry.Error OR tonG.Q THEN
                GVL_Mech.fbGantry.CmdExec := FALSE;
                aFailCode[6] := GVL_Mech.fbGantry.ErrorID; stp := 90;
            END_IF
        2: // sequence of targets 1, 3, 0
            CASE k OF 0: i := 1; 1: i := 3; 2: i := 0; END_CASE
            GVL_Mech.fbGridCar.TargetStation := i;
            GVL_Mech.fbGridCar.GotoExec := TRUE;
            tonG(IN := FALSE); stp := 3;
        3:
            IF GVL_Mech.fbGridCar.Done AND (GVL_Mech.fbGridCar.ActStation = i) THEN
                GVL_Mech.fbGridCar.GotoExec := FALSE;
                k := k + 1;
                IF k >= 3 THEN aResult[6] := 1; tc := 7; stp := 0;
                ELSE stp := 2; END_IF
            ELSIF GVL_Mech.fbGridCar.Error OR tonG.Q THEN
                GVL_Mech.fbGridCar.GotoExec := FALSE;
                aFailCode[6] := GVL_Mech.fbGridCar.ErrorID; stp := 90;
            END_IF
        90:
            aResult[6] := 2; tc := 7; stp := 0;
    END_CASE

// ================= TC7: fork fetch / return =================
7:
    CASE stp OF
        0:
            ptCur := T#40S; tonG(IN := FALSE);
            GVL_Mech.fbFork.Cmd.code := GVL_Cfg.MCMD_FETCH;
            GVL_Mech.fbFork.Cmd.p1 := 5.0;
            GVL_Mech.fbFork.CmdExec := TRUE;
            stp := 1;
        1:
            IF GVL_Mech.fbFork.Done AND GVL_Mech.fbFork.TrayHeld THEN
                GVL_Mech.fbFork.CmdExec := FALSE;
                GVL_Mech.fbFork.Cmd.code := GVL_Cfg.MCMD_RETURN;
                GVL_Mech.fbFork.Cmd.p1 := 5.0;
                tonG(IN := FALSE); stp := 12;   // one-scan gap for a real edge
            ELSIF GVL_Mech.fbFork.Error OR tonG.Q THEN
                GVL_Mech.fbFork.CmdExec := FALSE;
                aFailCode[7] := GVL_Mech.fbFork.ErrorID; stp := 90;
            END_IF
        12: // re-arm on a fresh scan
            GVL_Mech.fbFork.CmdExec := TRUE;
            stp := 2;
        2:
            IF GVL_Mech.fbFork.Done AND NOT GVL_Mech.fbFork.TrayHeld THEN
                GVL_Mech.fbFork.CmdExec := FALSE;
                aResult[7] := 1; tc := 8; stp := 0;
            ELSIF GVL_Mech.fbFork.Error OR tonG.Q THEN
                GVL_Mech.fbFork.CmdExec := FALSE;
                aFailCode[7] := GVL_Mech.fbFork.ErrorID; stp := 90;
            END_IF
        90:
            aResult[7] := 2; tc := 8; stp := 0;
    END_CASE

// ================= TC8: gantry pick / place / park =================
8:
    CASE stp OF
        0:
            ptCur := T#30S; tonG(IN := FALSE);
            GVL_Mech.fbGantry.Cmd.code := GVL_Cfg.MCMD_PICK;
            GVL_Mech.fbGantry.Cmd.p1 := 0.0;
            GVL_Mech.fbGantry.CmdExec := TRUE;
            stp := 1;
        1:
            IF GVL_Mech.fbGantry.Done AND GVL_Mech.fbGripper.Holding THEN
                GVL_Mech.fbGantry.CmdExec := FALSE;
                GVL_Mech.fbGantry.Cmd.code := GVL_Cfg.MCMD_PLACE;
                GVL_Mech.fbGantry.Cmd.p1 := 0.0;
                tonG(IN := FALSE); stp := 12;   // one-scan gap for a real edge
            ELSIF GVL_Mech.fbGantry.Error OR tonG.Q THEN
                GVL_Mech.fbGantry.CmdExec := FALSE;
                aFailCode[8] := GVL_Mech.fbGantry.ErrorID; stp := 90;
            END_IF
        2:
            IF GVL_Mech.fbGantry.Done AND NOT GVL_Mech.fbGripper.Holding THEN
                GVL_Mech.fbGantry.CmdExec := FALSE;
                GVL_Mech.fbGantry.Cmd.code := GVL_Cfg.MCMD_PARK;
                tonG(IN := FALSE); stp := 13;   // one-scan gap for a real edge
            ELSIF GVL_Mech.fbGantry.Error OR tonG.Q THEN
                GVL_Mech.fbGantry.CmdExec := FALSE;
                aFailCode[8] := GVL_Mech.fbGantry.ErrorID; stp := 90;
            END_IF
        12: // re-arm PLACE on a fresh scan
            GVL_Mech.fbGantry.CmdExec := TRUE;
            stp := 2;
        13: // re-arm PARK on a fresh scan
            GVL_Mech.fbGantry.CmdExec := TRUE;
            stp := 3;
        3:
            IF GVL_Mech.fbGantry.Done AND GVL_Mech.fbGantry.Parked THEN
                GVL_Mech.fbGantry.CmdExec := FALSE;
                aResult[8] := 1; tc := 9; stp := 0;
            ELSIF GVL_Mech.fbGantry.Error OR tonG.Q THEN
                GVL_Mech.fbGantry.CmdExec := FALSE;
                aFailCode[8] := GVL_Mech.fbGantry.ErrorID; stp := 90;
            END_IF
        90:
            aResult[8] := 2; tc := 9; stp := 0;
    END_CASE

// ================= TC9: full cycle via Gateway registers =================
9:
    CASE stp OF
        0: // enter RUN through the real path — but first wait for thermal readiness
           // (fridge pulldown / heat-up gate READY->RUN; on a fast suite run they
           //  may not be satisfied yet)
            GVL_Cmd.testMode := FALSE;
            haccp0 := GVL_Sts.haccpCount;
            ptCur := T#300S; tonG(IN := FALSE); stp := 30;
        30:
            IF GVL_Sts.heatAtSet AND GVL_Sts.fridgeAtSet AND GVL_Sts.allHomed THEN
                GVL_Cmd.reqStart := TRUE; holdCnt := 0;
                ptCur := T#20S; tonG(IN := FALSE); stp := 1;
            ELSIF tonG.Q THEN aFailCode[9] := 30; stp := 90; END_IF
        1:
            holdCnt := holdCnt + 1;
            IF holdCnt > 5 THEN GVL_Cmd.reqStart := FALSE; END_IF
            IF holdCnt > 10 THEN GVL_Cmd.reqStart := TRUE; holdCnt := 0; END_IF  // retry edge (one-shot may be rejected)
            IF GVL_Sts.mode = E_MachMode.RUN THEN
                GVL_Cmd.reqStart := FALSE; stp := 2;
            ELSIF tonG.Q THEN aFailCode[9] := 1; stp := 90; END_IF
        2: // FETCH_TRAY item=1 level=3 face=0
            testSeq := testSeq + 1;
            GVL_Cmd.mbCmdRegs[0] := testSeq;
            GVL_Cmd.mbCmdRegs[1] := GVL_Cfg.CMD_FETCH_TRAY;
            GVL_Cmd.mbCmdRegs[2] := 1;  GVL_Cmd.mbCmdRegs[3] := 0;   // p1 item
            GVL_Cmd.mbCmdRegs[4] := 3;  GVL_Cmd.mbCmdRegs[5] := 0;   // p2 level
            GVL_Cmd.mbCmdRegs[6] := 0;  GVL_Cmd.mbCmdRegs[7] := 0;   // p3 face
            ptCur := T#60S; tonG(IN := FALSE); stp := 3;
        3:
            IF (GVL_Cmd.gwAck.seqEcho = testSeq) AND GVL_Cmd.gwAck.done THEN stp := 4;
            ELSIF (GVL_Cmd.gwAck.seqEcho = testSeq) AND GVL_Cmd.gwAck.error THEN
                aFailCode[9] := GVL_Cmd.gwAck.errorId; stp := 90;
            ELSIF tonG.Q THEN aFailCode[9] := 3; stp := 90; END_IF
        4: // LOAD_GRIDDLE g=0 count=2 item=1
            testSeq := testSeq + 1;
            GVL_Cmd.mbCmdRegs[0] := testSeq;
            GVL_Cmd.mbCmdRegs[1] := GVL_Cfg.CMD_LOAD_GRIDDLE;
            GVL_Cmd.mbCmdRegs[2] := 0;  GVL_Cmd.mbCmdRegs[3] := 0;
            GVL_Cmd.mbCmdRegs[4] := 2;  GVL_Cmd.mbCmdRegs[5] := 0;
            GVL_Cmd.mbCmdRegs[6] := 1;  GVL_Cmd.mbCmdRegs[7] := 0;
            ptCur := T#120S; tonG(IN := FALSE); stp := 5;
        5:
            IF (GVL_Cmd.gwAck.seqEcho = testSeq) AND GVL_Cmd.gwAck.done THEN stp := 6;
            ELSIF (GVL_Cmd.gwAck.seqEcho = testSeq) AND GVL_Cmd.gwAck.error THEN
                aFailCode[9] := GVL_Cmd.gwAck.errorId; stp := 90;
            ELSIF tonG.Q THEN aFailCode[9] := 5; stp := 90; END_IF
        6: // wait cook done (90 s scaled by 5 -> ~18 s real)
            ptCur := T#120S; tonG(IN := FALSE); stp := 7;
        7:
            IF GVL_Sts.aGriddle[0].state = TO_UINT(E_GriddleState.READY_TO_SCRAPE) THEN stp := 8;
            ELSIF tonG.Q THEN aFailCode[9] := 7; stp := 90; END_IF
        8: // SCRAPE g=0
            testSeq := testSeq + 1;
            GVL_Cmd.mbCmdRegs[0] := testSeq;
            GVL_Cmd.mbCmdRegs[1] := GVL_Cfg.CMD_SCRAPE;
            GVL_Cmd.mbCmdRegs[2] := 0;  GVL_Cmd.mbCmdRegs[3] := 0;
            GVL_Cmd.mbCmdRegs[4] := 0;  GVL_Cmd.mbCmdRegs[6] := 0;
            ptCur := T#90S; tonG(IN := FALSE); stp := 9;
        9:
            IF (GVL_Cmd.gwAck.seqEcho = testSeq) AND GVL_Cmd.gwAck.done THEN stp := 10;
            ELSIF (GVL_Cmd.gwAck.seqEcho = testSeq) AND GVL_Cmd.gwAck.error THEN
                aFailCode[9] := GVL_Cmd.gwAck.errorId; stp := 90;
            ELSIF tonG.Q THEN aFailCode[9] := 9; stp := 90; END_IF
        10: // RETURN_TRAY level=3 face=0
            testSeq := testSeq + 1;
            GVL_Cmd.mbCmdRegs[0] := testSeq;
            GVL_Cmd.mbCmdRegs[1] := GVL_Cfg.CMD_RETURN_TRAY;
            GVL_Cmd.mbCmdRegs[2] := 3;  GVL_Cmd.mbCmdRegs[3] := 0;
            GVL_Cmd.mbCmdRegs[4] := 0;  GVL_Cmd.mbCmdRegs[5] := 0;
            ptCur := T#60S; tonG(IN := FALSE); stp := 11;
        11:
            IF (GVL_Cmd.gwAck.seqEcho = testSeq) AND GVL_Cmd.gwAck.done THEN
                // HACCP record must exist and be clean
                IF (GVL_Sts.haccpCount = haccp0 + 1) AND (GVL_Sts.lastHaccp.result = 0) THEN
                    aResult[9] := 1;
                ELSE
                    aResult[9] := 2; aFailCode[9] := 11;
                END_IF
                GVL_Cmd.testMode := TRUE;
                tc := 10; stp := 0;
            ELSIF (GVL_Cmd.gwAck.seqEcho = testSeq) AND GVL_Cmd.gwAck.error THEN
                aFailCode[9] := GVL_Cmd.gwAck.errorId; stp := 90;
            ELSIF tonG.Q THEN aFailCode[9] := 12; stp := 90; END_IF
        90:
            GVL_Cmd.testMode := TRUE;
            aResult[9] := 2; tc := 10; stp := 0;
    END_CASE

// ================= TC10: fault injection + recovery =================
10:
    CASE stp OF
        0: // inject: unreachable gantry target (idx 99 -> y >> arm)
            ptCur := T#30S; tonG(IN := FALSE);
            GVL_Mech.fbGantry.Cmd.code := GVL_Cfg.MCMD_PLACE;
            GVL_Mech.fbGantry.Cmd.p1 := 99.0;
            GVL_Mech.fbGantry.CmdExec := FALSE;  // may be left TRUE by JobExec (TC9) — force an edge
            stp := 20;
        20: // arm on a fresh scan
            GVL_Mech.fbGantry.CmdExec := TRUE;
            stp := 1;
        1:
            IF GVL_Mech.fbGantry.Error THEN
                GVL_Mech.fbGantry.CmdExec := FALSE;
                IF (GVL_Mech.fbGantry.ErrorID AND 16#FFFF) <> TO_UDINT(GVL_Cfg.ERR_UNREACH) THEN
                    aFailCode[10] := GVL_Mech.fbGantry.ErrorID; stp := 90;
                ELSE
                    tonG(IN := FALSE); stp := 2;
                END_IF
            ELSIF tonG.Q THEN aFailCode[10] := 1; stp := 90; END_IF
        2: // system must fall to FAULT via alarm cascade
            IF GVL_Sts.mode = E_MachMode.FAULT THEN
                GVL_Cmd.reqAckAll := TRUE; holdCnt := 0;
                tonG(IN := FALSE); stp := 3;
            ELSIF tonG.Q THEN aFailCode[10] := 2; stp := 90; END_IF
        3:
            holdCnt := holdCnt + 1;
            IF holdCnt > 5 THEN
                GVL_Cmd.reqAckAll := FALSE;
                GVL_Cmd.reqReset := TRUE; holdCnt := 0;
                stp := 4;
            END_IF
        4:
            holdCnt := holdCnt + 1;
            IF holdCnt > 5 THEN GVL_Cmd.reqReset := FALSE; END_IF
            IF holdCnt > 10 THEN GVL_Cmd.reqReset := TRUE; holdCnt := 0; END_IF  // retry edge
            IF GVL_Sts.mode = E_MachMode.HOMING THEN
                GVL_Cmd.reqReset := FALSE;
                ptCur := T#90S; tonG(IN := FALSE); stp := 5;
            ELSIF tonG.Q THEN aFailCode[10] := 4; stp := 90; END_IF
        5:
            IF (GVL_Sts.mode = E_MachMode.READY) AND GVL_Sts.allHomed THEN
                tonG(IN := FALSE); stp := 6;
            ELSIF tonG.Q THEN aFailCode[10] := 5; stp := 90; END_IF
        6: // inject 2: scraper sweep with interlock FALSE
            GVL_Mech.fbScraper.InterlockOk := FALSE;
            GVL_Mech.fbScraper.Cmd.code := GVL_Cfg.MCMD_SWEEP;
            GVL_Mech.fbScraper.Cmd.p1 := 0.0;
            GVL_Mech.fbScraper.CmdExec := TRUE;
            ptCur := T#20S; tonG(IN := FALSE); stp := 7;
        7:
            IF GVL_Mech.fbScraper.Error THEN
                GVL_Mech.fbScraper.CmdExec := FALSE;
                IF (GVL_Mech.fbScraper.ErrorID AND 16#FFFF) <> TO_UDINT(GVL_Cfg.ERR_INTERLOCK) THEN
                    aFailCode[10] := GVL_Mech.fbScraper.ErrorID; stp := 90;
                ELSE
                    tonG(IN := FALSE); stp := 8;
                END_IF
            ELSIF tonG.Q THEN aFailCode[10] := 7; stp := 90; END_IF
        8: // recover again
            IF GVL_Sts.mode = E_MachMode.FAULT THEN
                GVL_Cmd.reqAckAll := TRUE; holdCnt := 0; stp := 9;
            ELSIF tonG.Q THEN aFailCode[10] := 8; stp := 90; END_IF
        9:
            holdCnt := holdCnt + 1;
            IF holdCnt > 5 THEN
                GVL_Cmd.reqAckAll := FALSE;
                GVL_Cmd.reqReset := TRUE; holdCnt := 0;
                ptCur := T#90S; tonG(IN := FALSE); stp := 11;
            END_IF
        11:
            holdCnt := holdCnt + 1;
            IF holdCnt > 5 THEN GVL_Cmd.reqReset := FALSE; END_IF
            IF (holdCnt > 10) AND (GVL_Sts.mode = E_MachMode.FAULT) THEN
                GVL_Cmd.reqReset := TRUE; holdCnt := 0;   // retry edge while still faulted
            END_IF
            IF (GVL_Sts.mode = E_MachMode.READY) AND GVL_Sts.allHomed THEN
                GVL_Cmd.reqReset := FALSE;
                aResult[10] := 1; stp := 99;
            ELSIF tonG.Q THEN aFailCode[10] := 11; stp := 90; END_IF
        90:
            GVL_Mech.fbGantry.CmdExec := FALSE;
            GVL_Mech.fbScraper.CmdExec := FALSE;
            aResult[10] := 2; stp := 99;
        99: // ---- suite complete ----
            PassCount := 0;
            FOR i := 1 TO 10 DO
                IF aResult[i] = 1 THEN PassCount := PassCount + 1; END_IF
            END_FOR
            suiteDone := TRUE; running := FALSE;
            GVL_Cmd.testStart := FALSE;
    END_CASE
END_CASE

                  
END_PROGRAM

CONFIGURATION Device
  RESOURCE Application ON PLC
    VAR_GLOBAL CONSTANT  (* GVL_Cfg - ============================================================ GVL_Cfg — machine constants. VAR_GLOBAL CONSTANT. SIM_MODE is the ONLY switch between simulation and hardware. Set FALSE for production download. Never change at runtime. ============================================================ *)
      SIM_MODE : BOOL := TRUE;  (* <<< FALSE for real hardware *)
      SIM_TIME_SCALE : LREAL := 5.0;  (* thermal/cook acceleration in sim (1.0 = real time) *)
      T_MOTION_MS : LREAL := 4.0;
      T_APP_MS : LREAL := 20.0;
      GRIDDLE_COUNT : INT := 4;  (* ---- Counts & geometry ---- *)
      PATTIES_PER_GRIDDLE : INT := 6;
      STATIONS : INT := 4;  (* carousel stations *)
      STATION_LOAD : INT := 0;  (* station index where loading happens *)
      STATION_SCRAPE : INT := 2;  (* opposite station *)
      TRAY_COLS : INT := 6;
      TRAY_ROWS : INT := 4;
      PATTIES_PER_TRAY : INT := 24;
      TRAY_LEVELS : INT := 20;
      TRAY_FACES : INT := 2;
      ARM_LEN : LREAL := 350.0;  (* ---- Gantry kinematics (mm / deg) ---- *)
      GX_MIN : LREAL := 0.0;
      GX_MAX : LREAL := 900.0;
      THETA_MIN : LREAL := -90.0;
      THETA_MAX : LREAL := 90.0;
      GZ_UP : LREAL := 0.0;
      GZ_PICK : LREAL := 80.0;
      GZ_PLACE : LREAL := 60.0;
      THETA_SAFE : LREAL := 0.0;
      GX_PARK : LREAL := 50.0;
      PICK_BASE_X : LREAL := 700.0;  (* tray pick grid (chamber tray held by fork) *)
      PICK_BASE_Y : LREAL := -150.0;
      PICK_SPACING_X : LREAL := 60.0;
      PICK_SPACING_Y : LREAL := 60.0;
      PLACE_BASE_X : LREAL := 450.0;  (* griddle place grid (station 0, bottom platen) *)
      PLACE_BASE_Y : LREAL := 0.0;
      PLACE_SPC_X : LREAL := 70.0;
      PLACE_SPC_Y : LREAL := 70.0;
      PLACE_COLS : INT := 3;  (* 3 x 2 slots on a griddle *)
      G_VEL : LREAL := 400.0;  (* gantry X mm/s *)
      G_ACC : LREAL := 1500.0;  (* gantry X mm/s *)
      T_VEL : LREAL := 120.0;  (* theta deg/s *)
      T_ACC : LREAL := 500.0;  (* theta deg/s *)
      Z_VEL : LREAL := 200.0;
      Z_ACC : LREAL := 1000.0;
      S_VEL : LREAL := 300.0;  (* scraper *)
      S_ACC : LREAL := 1200.0;  (* scraper *)
      F_VEL : LREAL := 150.0;  (* fork *)
      F_ACC : LREAL := 400.0;  (* fork *)
      JOG_VEL_MAX : LREAL := 50.0;
      REC_COOK_MIN : LREAL := 10.0;  (* s *)
      REC_COOK_MAX : LREAL := 300.0;  (* s *)
      REC_SMDUR_MIN : LREAL := 0.0;  (* s *)
      REC_SMDUR_MAX : LREAL := 30.0;  (* s *)
      REC_SMPOS_MIN : LREAL := 2.0;  (* mm gap *)
      REC_SMPOS_MAX : LREAL := 12.0;  (* mm gap *)
      REC_HLPOS_MIN : LREAL := 3.0;  (* mm gap *)
      REC_HLPOS_MAX : LREAL := 15.0;  (* mm gap *)
      REC_PLSET_MIN : LREAL := 120.0;  (* degC *)
      REC_PLSET_MAX : LREAL := 230.0;  (* degC *)
      PRESS_OPEN_MM : LREAL := 60.0;  (* path 0 open position (clamshell gap) *)
      PRESS_TRIM_MAX_MM : LREAL := 2.0;  (* per-press calibration trim clamp (+/-) *)
      PRESS_BENCH_DRIVE : INT := 0;  (* bench: -1 = none; 0..3 = that press drive runs *)
      PRESS_PULSES_PER_MM : LREAL := 1000.0;  (* TODO calibrate: drive gear -> pulses per mm gap *)
      SC_ENGAGE_Z : LREAL := 45.0;  (* Channel setup reference (VERIFIED against CS2RS manual 5.4.1) — the registers live in the NetworkConfig channel config, not in code: write-multiple (FC16), length 2, per path: 0x6201 (path0 pos H/L), 0x6209 (path1), 0x6211 (path2). Trigger reg 0x6002 (unused; DI does motion). ---- Scraper geometry ---- *)
      SC_UP_Z : LREAL := 0.0;
      SC_SWEEP_X0 : LREAL := 100.0;
      SC_SWEEP_X1 : LREAL := 420.0;
      SC_ROW_Y : ARRAY[0..2] OF LREAL := [0.0, 70.0, 140.0];
      SC_STROKES : INT := 3;
      FORK_LEVEL_H : LREAL := 90.0;  (* mm per tray level *)
      FORK_Z0 : LREAL := 50.0;
      FORK_MICROLIFT : LREAL := 8.0;
      FORK_TELE_OUT : LREAL := 300.0;
      FORK_TELE_IN : LREAL := 0.0;
      ENC_CPR : DINT := 4096;  (* counts per carousel rev *)
      IDX_SPEED_FAST : INT := 300;  (* VFD speed ref (raw) *)
      IDX_SPEED_CREEP : INT := 40;
      IDX_DECEL_WIN : DINT := 300;  (* counts before target -> creep *)
      IDX_STOP_WIN : DINT := 25;  (* counts tolerance to drop pin *)
      IDX_VERIFY_WIN : DINT := 40;  (* encoder-vs-pin plausibility *)
      HEAT_ZONES : INT := 8;  (* ---- Heating ---- *)
      PWM_WINDOW_MS : LREAL := 2000.0;
      HEAT_KP : LREAL := 4.0;
      HEAT_KI : LREAL := 0.05;  (* %/ (degC*s) *)
      HEAT_AT_BAND : LREAL := 5.0;  (* |err| <= band -> atSet *)
      HEAT_MAX_STAGGER : INT := 2;  (* platens ramping at once *)
      TC_RATE_MAX : LREAL := 8.0;  (* degC/s plausibility *)
      FRIDGE_SET_C : LREAL := 4.0;
      FRIDGE_HYST_C : LREAL := 1.0;
      FRIDGE_EXC_S : LREAL := 300.0;  (* excursion > 5 min -> QUARANTINE *)
      TO_AXIS_MOVE : TIME := TIME#15s0ms;  (* ---- Timeouts ---- *)
      TO_AXIS_HOME : TIME := TIME#40s0ms;
      TO_PNEU : TIME := TIME#3s0ms;
      TO_PRESS : TIME := TIME#15s0ms;
      TO_INDEX : TIME := TIME#25s0ms;
      TO_MECH : TIME := TIME#1m0s0ms;
      SCRAPE_GUARD_S : LREAL := 8.0;
      GW_TIMEOUT_S : LREAL := 10.0;
      CMD_NOP : UINT := 0;  (* ---- Command codes: Gateway -> PLC (ST_GwCmd.code) ---- *)
      CMD_FETCH_TRAY : UINT := 1;  (* p1=item p2=level p3=face *)
      CMD_LOAD_GRIDDLE : UINT := 2;  (* p1=griddleId p2=count p3=item *)
      CMD_SCRAPE : UINT := 3;  (* p1=griddleId *)
      CMD_RETURN_TRAY : UINT := 4;  (* p1=level p2=face *)
      CMD_CLEAN_MODE : UINT := 5;
      CMD_ABORT : UINT := 6;
      MCMD_NONE : UINT := 0;  (* ---- Mechanism-local command codes (ST_MechCmd.code) ---- *)
      MCMD_HOME : UINT := 1;
      MCMD_PARK : UINT := 2;
      MCMD_PICK : UINT := 10;  (* gantry: p1=trayIdx(0..23) *)
      MCMD_PLACE : UINT := 11;  (* gantry: p1=slot(0..5) *)
      MCMD_SANITIZE : UINT := 13;
      MCMD_FETCH : UINT := 20;  (* fork: p1=level *)
      MCMD_RETURN : UINT := 21;  (* fork: p1=level *)
      MCMD_SWEEP : UINT := 30;  (* scraper: p1=strokeIdx(0..2) *)
      MCMD_PROFILE : UINT := 40;  (* press: recipe via SetRecipe inputs *)
      MCMD_OPEN : UINT := 41;  (* press open *)
      MCMD_GOTO : UINT := 50;  (* carousel: p1=station *)
      SS_GANTRY_X : UINT := 1;  (* ---- Subsystem IDs for ErrorID = SHL(ss,16) OR code ---- *)
      SS_GANTRY_T : UINT := 2;
      SS_GANTRY_Z : UINT := 3;
      SS_SCRAPER_X : UINT := 4;
      SS_SCRAPER_Y : UINT := 5;
      SS_SCRAPER_Z : UINT := 6;
      SS_FORK_Z : UINT := 7;
      SS_FORK_TELE : UINT := 8;
      SS_PRESS_0 : UINT := 10;  (* press n -> 10+n *)
      SS_GRID_CAR : UINT := 20;
      SS_FRIDGE_CAR : UINT := 21;
      SS_HEAT_0 : UINT := 30;  (* zone z -> 30+z *)
      SS_AIRLOCK : UINT := 40;
      SS_REFRIG : UINT := 41;
      SS_GANTRY : UINT := 45;
      SS_SCRAPER : UINT := 46;
      SS_FORK : UINT := 47;
      SS_GRIPPER : UINT := 48;
      SS_JOBEXEC : UINT := 50;
      SS_HOMING : UINT := 51;
      SS_GWCOMMS : UINT := 60;
      SS_PNEU : UINT := 61;
      SS_SENSOR : UINT := 62;
      ERR_NONE : UINT := 0;  (* ---- Generic error codes ---- *)
      ERR_TIMEOUT : UINT := 1;
      ERR_DRIVE : UINT := 2;
      ERR_NOT_HOMED : UINT := 3;
      ERR_UNREACH : UINT := 4;  (* IK unreachable *)
      ERR_BAD_CMD : UINT := 5;
      ERR_INTERLOCK : UINT := 6;
      ERR_PIN : UINT := 7;  (* pin/encoder mismatch *)
      ERR_SENSOR : UINT := 8;
      ERR_TC : UINT := 9;
      ERR_ABORTED : UINT := 10;
      ERR_BUSY : UINT := 11;
    END_VAR
    VAR_GLOBAL RETAIN  (* GVL_Par - ============================================================ GVL_Par — retained tunables (recipes, offsets). HMI-writable through bounds-checked paths only (PRG_HMI / PRG_GatewayComms). ============================================================ *)
      aRecipe : ARRAY[0..4] OF ST_Recipe := [(item := 0), (item := 1, cookTimeS := 90.0, smashDurS := 8.0, smashPosMm := 4.0, holdPosMm := 6.0, platenSetC := 200.0), (item := 2, cookTimeS := 110.0, smashDurS := 8.0, smashPosMm := 5.0, holdPosMm := 7.0, platenSetC := 200.0), (item := 3, cookTimeS := 60.0, smashDurS := 0.0, smashPosMm := 8.0, holdPosMm := 8.0, platenSetC := 190.0), (item := 4, cookTimeS := 45.0, smashDurS := 0.0, smashPosMm := 8.0, holdPosMm := 8.0, platenSetC := 180.0)];  (* Index by E_Item value 0..4; [0] unused *)
      jogVel : LREAL := 20.0;  (* PINEAPPLE *)
      pickOffsetX : LREAL := 0.0;  (* commissioning trims *)
      pickOffsetY : LREAL := 0.0;
      placeOffsetX : LREAL := 0.0;
      placeOffsetY : LREAL := 0.0;
      pressTrimMm : ARRAY[0..3] OF LREAL := [0.0, 0.0, 0.0, 0.0];  (* per-press smash/hold position trim, mm (+ = larger gap); HMI-adjustable, clamped to +/- GVL_Cfg.PRESS_TRIM_MAX_MM in PRG_HMI *)
    END_VAR
    VAR_GLOBAL  (* GVL_IO - ============================================================ GVL_IO — the ONLY POU with physical addresses. SIM NOTE: in SIM_MODE these are never read/written (PRG_IoMap short-circuits). Addresses below are PLACEHOLDERS — replace with the real electrical map during panel design (see MIGRATION_GUIDE.md step 2) and keep wire numbers in comments. ============================================================ *)
      qPressSel0 : ARRAY[0..3] OF BOOL;  (* TODO real per-drive addresses *)
      qPressSel1 : ARRAY[0..3] OF BOOL;
      qPressCtrg : ARRAY[0..3] OF BOOL;
      qPressEnable : ARRAY[0..3] OF BOOL;
      iPressInPos : ARRAY[0..3] OF BOOL;
      iPressAlarm : ARRAY[0..3] OF BOOL;
      qDoorFridgeFront AT %QX4.0 : BOOL;  (* ---- Pneumatics ---- *)
      qDoorFridgeSide AT %QX4.1 : BOOL;
      qDoorChamber AT %QX4.2 : BOOL;
      qPinGriddle AT %QX4.3 : BOOL;
      qPinFridge AT %QX4.4 : BOOL;
      qGripper AT %QX4.5 : BOOL;
      iDoorFrFront_Op AT %IX3.0 : BOOL;
      iDoorFrFront_Cl AT %IX3.1 : BOOL;
      iDoorFrSide_Op AT %IX3.2 : BOOL;
      iDoorFrSide_Cl AT %IX3.3 : BOOL;
      iDoorChamber_Op AT %IX3.4 : BOOL;
      iDoorChamber_Cl AT %IX3.5 : BOOL;
      iPinGriddle_Ext AT %IX3.6 : BOOL;
      iPinGriddle_Ret AT %IX3.7 : BOOL;
      iPinFridge_Ext AT %IX4.0 : BOOL;
      iPinFridge_Ret AT %IX4.1 : BOOL;
      iGripAcquired AT %IX4.2 : BOOL;
      qGridCarFwd AT %QX5.0 : BOOL;  (* ---- Carousel VFDs (hardwired run/dir + analog/comms speed) ---- *)
      qGridCarRev AT %QX5.1 : BOOL;
      qFrCarFwd AT %QX5.2 : BOOL;
      qFrCarRev AT %QX5.3 : BOOL;
      wGridCarSpeed AT %QW10 : INT;
      wFrCarSpeed AT %QW11 : INT;
      diGridCarEnc AT %ID12 : DINT;
      diFrCarEnc AT %ID14 : DINT;
      iGridCarHome AT %IX5.0 : BOOL;
      iFrCarHome AT %IX5.1 : BOOL;
      qSsr : ARRAY[0..7] OF BOOL;  (* ---- Heating (R2 modules) ---- *)
      wPlatenTemp AT %IW20 : ARRAY[0..7] OF INT;  (* 0.1 degC *)
      wFridgeTemp AT %IW28 : INT;  (* 0.1 degC *)
      qBenchPrAdd0 AT %QX1.5 : BOOL;  (* drive SI = ADD0 (ex Z_DO_Down) *)
      qBenchPrAdd1 AT %QX1.7 : BOOL;  (* drive SI = ADD1 (ex end_effector — VERIFY wire + SI assign) *)
      qBenchPrCtrg AT %QX1.6 : BOOL;  (* drive SI = CTRG (ex Z_Trig) *)
      qBenchPrDisable AT %QX1.3 : BOOL;  (* drive enable line, INVERTED: TRUE = disable (ex Z_Disable) *)
      iBenchPrInPos AT %IX1.0 : BOOL;  (* SO1 INP (ex Z_InPos) *)
      iBenchPrAlarm AT %IX1.1 : BOOL;  (* SO3 ALM (ex Z_Alarm — check polarity!) *)
      qMbPr0Data AT %QW49 : ARRAY[0..1] OF WORD;  (* CH0: slave1 FC16 25089/0x6201 len2 (path0 pos H,L) *)
      qMbPr1Data AT %QW52 : ARRAY[0..1] OF WORD;  (* CH1: slave1 FC16 25097/0x6209 len2 (path1) *)
      qMbPr2Data AT %QW55 : ARRAY[0..1] OF WORD;  (* CH2: slave1 FC16 25105/0x6211 len2 (path2) *)
      qMbPr0Trig AT %QX102.0 : BOOL;  (* trigger control bits *)
      qMbPr1Trig AT %QX108.0 : BOOL;
      qMbPr2Trig AT %QX114.0 : BOOL;
      iMbPr0Done AT %IX198.0 : BOOL;  (* processing complete states *)
      iMbPr1Done AT %IX198.1 : BOOL;
      iMbPr2Done AT %IX198.2 : BOOL;
      iMbPrErr AT %IW98 : WORD;  (* master ErrorCode (0 = ok) *)
      qForkBrakeRelease AT %QX7.0 : BOOL;  (* ---- Fork brake ---- *)
      iForkBrakeOk AT %IX6.0 : BOOL;
      iForkTrayPresent AT %IX6.1 : BOOL;
      iSafetyOk AT %IX7.0 : BOOL;  (* ---- Safety controller status (monitor only) ---- *)
      iZonePwrMotion AT %IX7.1 : BOOL;
      iZonePwrPress AT %IX7.2 : BOOL;
    END_VAR
    VAR_GLOBAL  (* GVL_Axes - ============================================================ GVL_Axes — SoftMotion axis references. SIMULATION BUILD: the dummy declarations below let the project compile with SM3_Basic present but no drives; FB_AxisCtrl never calls MC_* while SIM_MODE=TRUE. PRODUCTION BUILD: DELETE these dummies and pass the device-tree axis objects (names created by the EtherCAT config) directly in PRG_Motion — see MIGRATION_GUIDE.md step 3. ============================================================ *)
      axRefGantryX : AXIS_REF_SM3;
      axRefGantryT : AXIS_REF_SM3;
      axRefGantryZ : AXIS_REF_SM3;
      axRefScraperX : AXIS_REF_SM3;
      axRefScraperY : AXIS_REF_SM3;
      axRefScraperZ : AXIS_REF_SM3;
      axRefForkZ : AXIS_REF_SM3;
      axRefForkTele : AXIS_REF_SM3;
    END_VAR
    VAR_GLOBAL  (* GVL_Cmd - ============================================================ GVL_Cmd — commands INTO the PLC (Gateway + HMI + test). Modbus-TCP register images live here (%MW). The MC508 Modbus TCP slave exposes %MW to the Gateway. ============================================================ *)
      mbCmdRegs AT %MW0 : ARRAY[0..9] OF WORD;  (* seq,code,p1..p4 (DINT lo/hi) *)
      mbAckRegs AT %MW10 : ARRAY[0..5] OF WORD;
      mbStsRegs AT %MW20 : ARRAY[0..79] OF WORD;
      mbParRegs AT %MW500 : ARRAY[0..59] OF WORD;
      gwCmd : ST_GwCmd;  (* decoded, latched command *)
      gwAck : ST_GwAck;
      gwHeartbeatIn : UINT;  (* written by Gateway (reg in mbCmdRegs[9]) *)
      gwAlive : BOOL;
      gwPending : BOOL;  (* new latched command awaiting JobExec *)
      hmiStart : BOOL;  (* HMI request bits (edge-processed in PRG_HMI) *)
      hmiStop : BOOL;
      hmiReset : BOOL;
      hmiAck : BOOL;
      hmiClean : BOOL;
      hmiMaintPin : UINT;  (* maintenance password value *)
      hmiJogAxis : INT;  (* 0=none 1..8 *)
      hmiJogPlus : BOOL;
      hmiJogMinus : BOOL;
      hmiRecItem : UINT;  (* 1..4 = E_Item to edit *)
      hmiRecField : UINT;  (* 1=cookTimeS 2=smashDurS 3=smashPosMm 4=holdPosMm 5=platenSetC *)
      hmiRecValue : LREAL;  (* requested value *)
      hmiRecWrite : BOOL;  (* rising edge applies *)
      hmiRecAck : BOOL;  (* feedback: accepted *)
      hmiRecErr : BOOL;  (* feedback: rejected (bounds / mode / index) *)
      hmiTrimPress : UINT;  (* 0..3 *)
      hmiTrimDelta : LREAL;  (* +/- mm added to that press's trim *)
      hmiTrimWrite : BOOL;  (* rising edge applies *)
      hmiTrimAck : BOOL;
      hmiTrimErr : BOOL;
      hmiRegsCmd AT %MW600 : ARRAY[0..9] OF WORD;  (* LT2100E Modbus-TCP register image (see HMI_LT2100E_GUIDE.md) HMI writes 600..609, reads 620..669. Packed/unpacked in PRG_HMI. *)
      hmiRegsSts AT %MW620 : ARRAY[0..49] OF WORD;
      reqStart : BOOL;  (* Processed requests to Supervisor *)
      reqStop : BOOL;
      reqReset : BOOL;
      reqClean : BOOL;
      reqAckAll : BOOL;
      testMode : BOOL := TRUE;  (* default TRUE in sim; set FALSE for gateway runs *)
      testStart : BOOL;  (* rising edge starts the automated suite *)
    END_VAR
    VAR_GLOBAL  (* GVL_Sts - ============================================================ GVL_Sts — status OUT of the PLC + Supervisor coordination flags. Written by L2/L3 only; L4 reads. ============================================================ *)
      mode : E_MachMode := E_MachMode.BOOT;
      uptimeS : UDINT;
      heartbeat : UINT;
      safetyOk : BOOL;  (* effective (sim: TRUE) *)
      enMotion : BOOL;  (* mechanisms may move *)
      enProcess : BOOL;  (* heat + refrigeration on *)
      abortAll : BOOL;  (* broadcast abort *)
      resetPulse : BOOL;  (* 1-cycle axis reset on FAULT->HOMING *)
      cleanCoolOk : BOOL;  (* all platens < 60 C in CLEAN *)
      allHomed : BOOL;  (* Aggregates *)
      heatAtSet : BOOL;
      fridgeAtSet : BOOL;
      fridgeActC : LREAL;
      aGriddle : ARRAY[0..3] OF ST_GriddleSts;
      aHeat : ARRAY[0..7] OF ST_HeatZone;
      tray : ST_TrayInfo;
      pattyOnGriddle : ARRAY[0..3, 0..5] OF BOOL;  (* process bookkeeping (v1: no optics) *)
      carGridStation : INT;
      carFridgeFace : INT;
      haccpCount : UDINT;
      lastHaccp : ST_HaccpRec;
      activeAlarms : INT;
      gwSilent : BOOL;
    END_VAR
    VAR_GLOBAL  (* GVL_Alm - ============================================================ GVL_Alm — alarm table + history. Managed by PRG_Alarms and F_RaiseAlarm (any POU may raise). ============================================================ *)
      aActive : ARRAY[0..63] OF ST_Alarm;
      nActive : INT;
      worstClass : UINT;  (* highest active E_FaultClass *)
      reqZoneStop : BOOL;  (* aggregated flags for Supervisor *)
      reqMachStop : BOOL;
      aHistory : ARRAY[0..199] OF ST_Alarm;
      histHead : INT;
    END_VAR
    VAR_GLOBAL  (* GVL_Mech - ============================================================ GVL_Mech — ALL FB instances live here (single ownership table). BODY-CALL OWNERSHIP (call the FB body ONLY in the listed PRG): PRG_Motion (T_Motion): axis FBs, fbGantry, fbScraper, fbFork, fbGripper PRG_Carousels(T_App) : press drives, presses, VFDs, carousels, pneumatics, airlock PRG_Heating (T_App) : heaters, heat bank, refrigeration All other POUs only WRITE inputs / READ outputs of these instances. ============================================================ *)
      axGX : FB_AxisCtrl;  (* gantry X / theta / Z *)
      axGT : FB_AxisCtrl;  (* gantry X / theta / Z *)
      axGZ : FB_AxisCtrl;  (* gantry X / theta / Z *)
      axSX : FB_AxisCtrl;  (* scraper *)
      axSY : FB_AxisCtrl;  (* scraper *)
      axSZ : FB_AxisCtrl;  (* scraper *)
      axFZ : FB_AxisCtrl;  (* fork Z / telescope *)
      axFT : FB_AxisCtrl;  (* fork Z / telescope *)
      drvPress : ARRAY[0..3] OF FB_PressDrive;  (* L1 press drives + L2 presses *)
      fbPress : ARRAY[0..3] OF FB_Press;
      fbDoorFridgeFront : FB_PneuActuator;  (* Pneumatics *)
      fbDoorFridgeSide : FB_PneuActuator;
      fbDoorChamber : FB_PneuActuator;
      fbPinGriddle : FB_PneuActuator;
      fbPinFridge : FB_PneuActuator;
      fbPneuGrip : FB_PneuActuator;
      vfdGriddle : FB_VfdIndex;  (* Carousels *)
      vfdFridge : FB_VfdIndex;
      fbGridCar : FB_GriddleCarousel;
      fbFridgeCar : FB_FridgeCarousel;
      fbHeater : ARRAY[0..7] OF FB_PidHeater;  (* Heating / cold *)
      fbHeatBank : FB_HeatBank;
      fbRefrig : FB_Refrigeration;
      fbIK : FB_IKTransform;  (* Motion mechanisms *)
      fbGripper : FB_Gripper;
      fbGantry : FB_Gantry;
      fbScraper : FB_Scraper;
      fbFork : FB_Fork;
      fbAirlock : FB_Airlock;  (* Coordination *)
      fbHoming : FB_HomingManager;
      fbTracker : FB_GriddleTracker;
      fbQueue : FB_JobQueue;
    END_VAR
    TASK T_Motion(INTERVAL := T#4ms, PRIORITY := 1);
    TASK T_App(INTERVAL := T#20ms, PRIORITY := 8);
    TASK EtherCAT_Master_Leadshine_A(INTERVAL := T#4ms, PRIORITY := 0);
    TASK T_Comms(INTERVAL := T#100ms, PRIORITY := 15);
    PROGRAM PRG_Motion WITH T_Motion : PRG_Motion;
    PROGRAM PRG_IoMap WITH T_App : PRG_IoMap;
    PROGRAM PRG_Supervisor WITH T_App : PRG_Supervisor;
    PROGRAM PRG_JobExec WITH T_App : PRG_JobExec;
    PROGRAM PRG_Test WITH T_App : PRG_Test;
    PROGRAM PRG_Carousels WITH T_App : PRG_Carousels;
    PROGRAM PRG_Heating WITH T_App : PRG_Heating;
    PROGRAM PRG_Sim WITH T_App : PRG_Sim;
    PROGRAM PRG_Alarms WITH T_App : PRG_Alarms;
    PROGRAM EtherCAT_Master_Leadshine_A.EtherCAT_Task WITH EtherCAT_Master_Leadshine_A : EtherCAT_Master_Leadshine_A.EtherCAT_Task;
    PROGRAM PRG_GatewayComms WITH T_Comms : PRG_GatewayComms;
    PROGRAM PRG_HMI WITH T_Comms : PRG_HMI;
    PROGRAM PRG_HACCP WITH T_Comms : PRG_HACCP;
  END_RESOURCE
END_CONFIGURATION

CONFIGURATION High_Speed_IO_Module
END_CONFIGURATION

CONFIGURATION LocalBus_Master_Module
END_CONFIGURATION

CONFIGURATION EtherCAT_Master_Leadshine_A
END_CONFIGURATION

CONFIGURATION CS3E_D1008
END_CONFIGURATION

CONFIGURATION Axis
END_CONFIGURATION

CONFIGURATION CS3E_D1008_1
END_CONFIGURATION

CONFIGURATION Axis_1
END_CONFIGURATION

CONFIGURATION CS3E_D1008_2
END_CONFIGURATION

CONFIGURATION Axis_2
END_CONFIGURATION

CONFIGURATION CS3E_D1008_3
END_CONFIGURATION

CONFIGURATION Axis_3
END_CONFIGURATION

CONFIGURATION CS3E_D1008_4
END_CONFIGURATION

CONFIGURATION Axis_4
END_CONFIGURATION

CONFIGURATION CS3E_D1008_5
END_CONFIGURATION

CONFIGURATION Axis_5
END_CONFIGURATION

CONFIGURATION CS3E_D1008_6
END_CONFIGURATION

CONFIGURATION Axis_6
END_CONFIGURATION

CONFIGURATION CS3E_D1008_7
END_CONFIGURATION

CONFIGURATION Axis_7
END_CONFIGURATION

CONFIGURATION ModbusCOM_Master_1
END_CONFIGURATION

CONFIGURATION ModbusCOM_Slave
END_CONFIGURATION

CONFIGURATION ModbusCOM_Slave_1
END_CONFIGURATION

CONFIGURATION ModbusCOM_Slave_2
END_CONFIGURATION

CONFIGURATION ModbusCOM_Slave_3
END_CONFIGURATION

CONFIGURATION ModbusTCP_Slave_Device
END_CONFIGURATION

CONFIGURATION SoftMotion General Axis Pool
END_CONFIGURATION
